// TIA Portal V18 export
DATA_BLOCK "SS2_A1_8RTD_AI_Vars"   // DB11121
{ S7_Optimized_Access := 'FALSE' }
VERSION : 0.1
// stored: AutoNumber false, DBAccessibleFromOPCUA true, IsOnlyStoredInLoadMemory false, IsWriteProtectedInAS false
   VAR
      AI1 { S7_SetPoint := 'True'} : "UDT_RTDadv";
      AI2 { S7_SetPoint := 'True'} : "UDT_RTDadv";
      AI3 { S7_SetPoint := 'True'} : "UDT_RTDadv";
      AI4 { S7_SetPoint := 'True'} : "UDT_RTDadv";
      AI5 { S7_SetPoint := 'True'} : "UDT_RTDadv";
      AI6 { S7_SetPoint := 'True'} : "UDT_RTDadv";
      AI7 { S7_SetPoint := 'True'} : "UDT_RTDadv";
      AI8 { S7_SetPoint := 'True'} : "UDT_RTDadv";
   END_VAR
BEGIN
   AI1.cFuncSystemID := 2;
   AI1.cFuncVar := 6;
   AI2.cFuncSystemID := 2;
   AI2.cFuncVar := 4;
   AI3.cFuncSystemID := 2;
   AI3.cFuncVar := 3;
   AI4.cFuncSystemID := 10;
   AI4.cFuncVar := 3;
   AI5.cFuncSystemID := 10;
   AI5.cFuncVar := 5;
   AI6.cFuncSystemID := 10;
   AI6.cFuncVar := 6;
   AI7.cFuncSystemID := 10;
   AI7.cFuncVar := 8;
   AI8.cFuncSystemID := 10;
   AI8.cFuncVar := 9;
END_DATA_BLOCK
